// TIA Portal V19 export
FUNCTION_BLOCK "Pendant_FB"   // FB77, LAD
// stored: Access Published, MemoryReserve 100, SetENOAutomatically false
   VAR_INPUT
      SwitchEnable : Bool := TRUE;   // Put your PB interlocking conditions in here.
      Command : Bool;   // Put your Two hands command or Jog+ and Jog- commands in parallel.
      "Jog+" : Bool;   // Put your Jog+ selection or command in here.
      "Jog-" : Bool;   // Put your Jog- selection or command in here.
   END_VAR
   VAR_OUTPUT
      "Action+" : Bool;
      "Action-" : Bool;
      SelectionPE : Bool;
      ResetAlm : Bool;   // Job+ & Jog- & !Command
   END_VAR
   VAR DB_SPECIFIC
      "Jog+Lp" : Bool;
      "Jog-Lp" : Bool;
   END_VAR
BEGIN

REGION Network 1: One Shot Selection
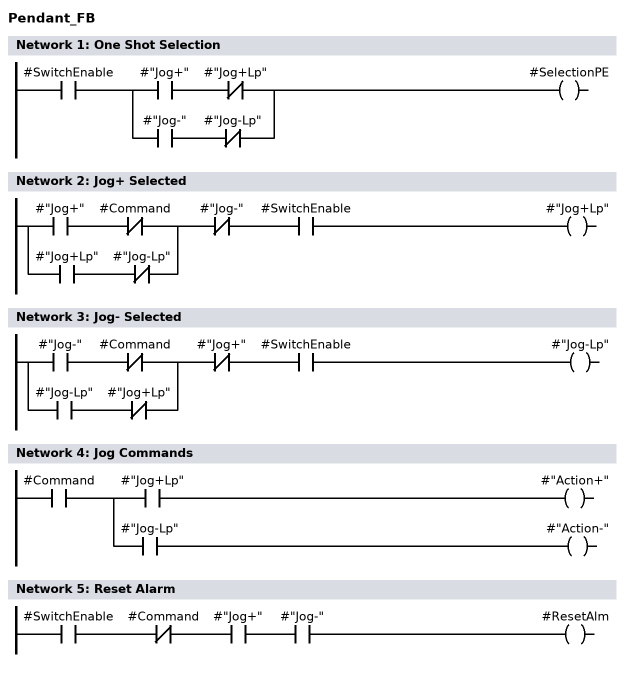
   RUNG wire#powerrail
      Contact( #SwitchEnable )
      wire#w1
      Contact( #"Jog+" )
      I_Contact( #"Jog+Lp" )
      wire#w2
      Coil( #SelectionPE )
   END_RUNG
   RUNG wire#w1
      Contact( #"Jog-" )
      I_Contact( #"Jog-Lp" )
   END_RUNG wire#w2
   // the same network as SCL:
   #SelectionPE := #SwitchEnable AND ((#"Jog+" AND NOT #"Jog+Lp") OR (#"Jog-" AND NOT #"Jog-Lp"));
END_REGION

REGION Network 2: Jog+ Selected
   RUNG wire#powerrail
      Contact( #"Jog+" )
      I_Contact( #Command )
      wire#w1
      I_Contact( #"Jog-" )
      Contact( #SwitchEnable )
      Coil( #"Jog+Lp" )
   END_RUNG
   RUNG wire#powerrail
      Contact( #"Jog+Lp" )
      I_Contact( #"Jog-Lp" )
   END_RUNG wire#w1
   // the same network as SCL:
   #"Jog+Lp" := ((#"Jog+" AND NOT #Command) OR (#"Jog+Lp" AND NOT #"Jog-Lp")) AND NOT #"Jog-" AND #SwitchEnable;
END_REGION

REGION Network 3: Jog- Selected
   RUNG wire#powerrail
      Contact( #"Jog-" )
      I_Contact( #Command )
      wire#w1
      I_Contact( #"Jog+" )
      Contact( #SwitchEnable )
      Coil( #"Jog-Lp" )
   END_RUNG
   RUNG wire#powerrail
      Contact( #"Jog-Lp" )
      I_Contact( #"Jog+Lp" )
   END_RUNG wire#w1
   // the same network as SCL:
   #"Jog-Lp" := ((#"Jog-" AND NOT #Command) OR (#"Jog-Lp" AND NOT #"Jog+Lp")) AND NOT #"Jog+" AND #SwitchEnable;
END_REGION

REGION Network 4: Jog Commands
   RUNG wire#powerrail
      Contact( #Command )
      wire#w1
      Contact( #"Jog+Lp" )
      Coil( #"Action+" )
   END_RUNG
   RUNG wire#w1
      Contact( #"Jog-Lp" )
      Coil( #"Action-" )
   END_RUNG
   // the same network as SCL:
   #"Action+" := #Command AND #"Jog+Lp";
   #"Action-" := #Command AND #"Jog-Lp";
END_REGION

REGION Network 5: Reset Alarm
   RUNG wire#powerrail
      Contact( #SwitchEnable )
      I_Contact( #Command )
      Contact( #"Jog+" )
      Contact( #"Jog-" )
      Coil( #ResetAlm )
   END_RUNG
   // the same network as SCL:
   #ResetAlm := #SwitchEnable AND NOT #Command AND #"Jog+" AND #"Jog-";
END_REGION
END_FUNCTION_BLOCK
